// TIA Portal V20 export
FUNCTION_BLOCK "Side_Shifters"   // FB12, LAD
{ S7_Optimized_Access := 'TRUE' }
// stored: MemoryReserve 100, SetENOAutomatically false
   VAR_INPUT
      set_Hydraulic_Up { ExternalAccessible := 'False'; ExternalVisible := 'False'; ExternalWritable := 'False'} : Bool;
      set_Hydraulic_Down { ExternalAccessible := 'False'; ExternalVisible := 'False'; ExternalWritable := 'False'} : Bool;
      set_SL_Hydraulic_Up : Bool;
      set_SL_Hydraulic_Down : Bool;
      set_SR_Hydraulic_Up : Bool;
      set_SR_Hydraulic_Down : Bool;
      set_SL_Hydraulic_Unit : Bool;
      set_SR_Hydraulic_Unit : Bool;
      set_Go_To_ST1 : Bool;
      set_Go_To_ST2 : Bool;
      set_Go_To_ST3 : Bool;
      set_Go_To_ST4 : Bool;
      ST1_Empty : Bool;
      ST2_Empty : Bool;
      ST3_Empty : Bool;
      ST4_Empty : Bool;
      Homing_1_SR : Int;
      Homing_2_SR : Int;
      Homing_3_SR : Int;
      Homing_4_SR : Int;
      Homing_1_SL : Int;
      Homing_2_SL : Int;
      Homing_3_SL : Int;
      Homing_4_SL : Int;
      SL_Drive_Forward : Bool;
      SL_Drive_Backward : Bool;
      SR_Drive_Forward : Bool;
      SR_Drive_Backward : Bool;
      iSL_Sen_Drv_1 : Bool;
      iSL_Sen_Drv_2 : Bool;
      iSL_Sen_Drv_3 : Bool;
      iSL_Sen_Drv_4 : Bool;
      iSR_Sen_Drv_1 : Bool;
      iSR_Sen_Drv_2 : Bool;
      iSR_Sen_Drv_3 : Bool;
      iSR_Sen_Drv_4 : Bool;
      iSL_Sen_Val1_Up : Bool;
      iSL_Sen_Val1_Down : Bool;
      iSL_Sen_Val2_Up : Bool;
      iSL_Sen_Val2_Down : Bool;
      iSR_Sen_Val1_Up : Bool;
      iSR_Sen_Val1_Down : Bool;
      iSR_Sen_Val2_Up : Bool;
      iSR_Sen_Val2_Down : Bool;
      iSL_Distance : Int;
      iSR_Correct : Int;
      iSR_Distance : Int;
      iSL_Hydraulic_Filtr : Bool;
      iSR_Hydraulic_Empty : Bool;
      HWIdentSL : HW_IO;
      HWIdentSR : HW_IO;
      Reset_Drive : Bool;
      Reset_Hydro : Bool;
   END_VAR
   VAR_OUTPUT
      oSL_Valve_Up { ExternalAccessible := 'False'; ExternalVisible := 'False'; ExternalWritable := 'False'} : Bool;
      oSL_Valve_Down { ExternalAccessible := 'False'; ExternalVisible := 'False'; ExternalWritable := 'False'} : Bool;
      oSL_Hydraulic_Unit { ExternalAccessible := 'False'; ExternalVisible := 'False'; ExternalWritable := 'False'} : Bool;
      oSR_Valve_Up { ExternalAccessible := 'False'; ExternalVisible := 'False'; ExternalWritable := 'False'} : Bool;
      oSR_Valve_Down { ExternalAccessible := 'False'; ExternalVisible := 'False'; ExternalWritable := 'False'} : Bool;
      oSR_Hydraulic_Unit { ExternalAccessible := 'False'; ExternalVisible := 'False'; ExternalWritable := 'False'} : Bool;
      oHydraulic_Status_LED_UP_1 : Bool;
      oHydraulic_Status_LED_UP_2 : Bool;
      oHydraulic_Status_LED_DOWN_1 : Bool;
      oHydraulic_Status_LED_DOWN_2 : Bool;
      oSL_Communication_OK : Bool;
      oSR_Communication_OK : Bool;
      oSL_Forward_Flag : Bool;
      oSL_Backward_Flag : Bool;
      oSR_Forward_Flag : Bool;
      oSR_Backward_Flag : Bool;
      oST1_1_Move_Flag : Bool;
      oST1_2_Move_Flag : Bool;
      oST2_1_Move_Flag : Bool;
      oST2_2_Move_Flag : Bool;
      oST3_1_Move_flag : Bool;
      oST3_2_Move_Flag : Bool;
      oST4_1_Move_Flag : Bool;
      oST4_2_Move_Flag : Bool;
   END_VAR
   VAR_IN_OUT
      iSL_Drive_Param : "SEW_MOVIKIT_VelocityDrive_STATUS_V2.1";
      iSR_Drive_Param : "SEW_MOVIKIT_VelocityDrive_STATUS_V2.1";
      oSL_Drive_Param : "SEW_MOVIKIT_VelocityDrive_SETPOINTS_V2.1";
      oSR_Drive_Param : "SEW_MOVIKIT_VelocityDrive_SETPOINTS_V2.1";
   END_VAR
   VAR
      Hydraulic_SL { ExternalAccessible := 'False'; ExternalVisible := 'False'; ExternalWritable := 'False'} : "Side_Hydraulic";
      Hydraulic_SR { ExternalAccessible := 'False'; ExternalVisible := 'False'; ExternalWritable := 'False'} : "Side_Hydraulic";
      Side_Driver_Instance { S7_SetPoint := 'True'} : "Side_Driver";
      Side_Shifter_Auto_Instance { S7_SetPoint := 'True'} : "Side_Shifter_Auto";
      SL_Auto_Speed { S7_SetPoint := 'True'} : Int := 1000;
      SR_Auto_Speed { S7_SetPoint := 'True'} : Int := 1000;
      SL_Auto_Forward : Bool;
      SL_Auto_Backward : Bool;
      SR_Auto_Forward : Bool;
      SR_Auto_Backward : Bool;
      SR_Distance_Correct : Int;
      SL_Error_Laser : Bool;
      SR_Error_Laser : Bool;
      SL_SR_InPosition : Bool;
      SL_Sen_Up : Bool;
      SL_Sen_Down : Bool;
      SR_Sen_Up : Bool;
      SR_Sen_Down : Bool;
      SL_Error_Hyd : Bool;
      SR_Error_Hyd : Bool;
      Error_Drive : Bool;
      Error_Hydro : Bool;
      Status_Sen_Up : Bool;
      Status_Sen_Down : Bool;
      RL_Speed : Int;
      RR_Speed : Int;
      Step_Move_Pallets : Int;
      Row_Start : Int;
      Row_Destination : Int;
      Column_Start : Int;
      Column_Destination : Int;
      TON_iSR_Error { S7_SetPoint := 'True'} : TON_TIME;
      TON_iSL_Error { S7_SetPoint := 'True'} : TON_TIME;
   END_VAR
   VAR_TEMP
      i : SInt;
      FoundIndex : SInt;
   END_VAR
BEGIN

REGION Network 1: Hydraulic control SL
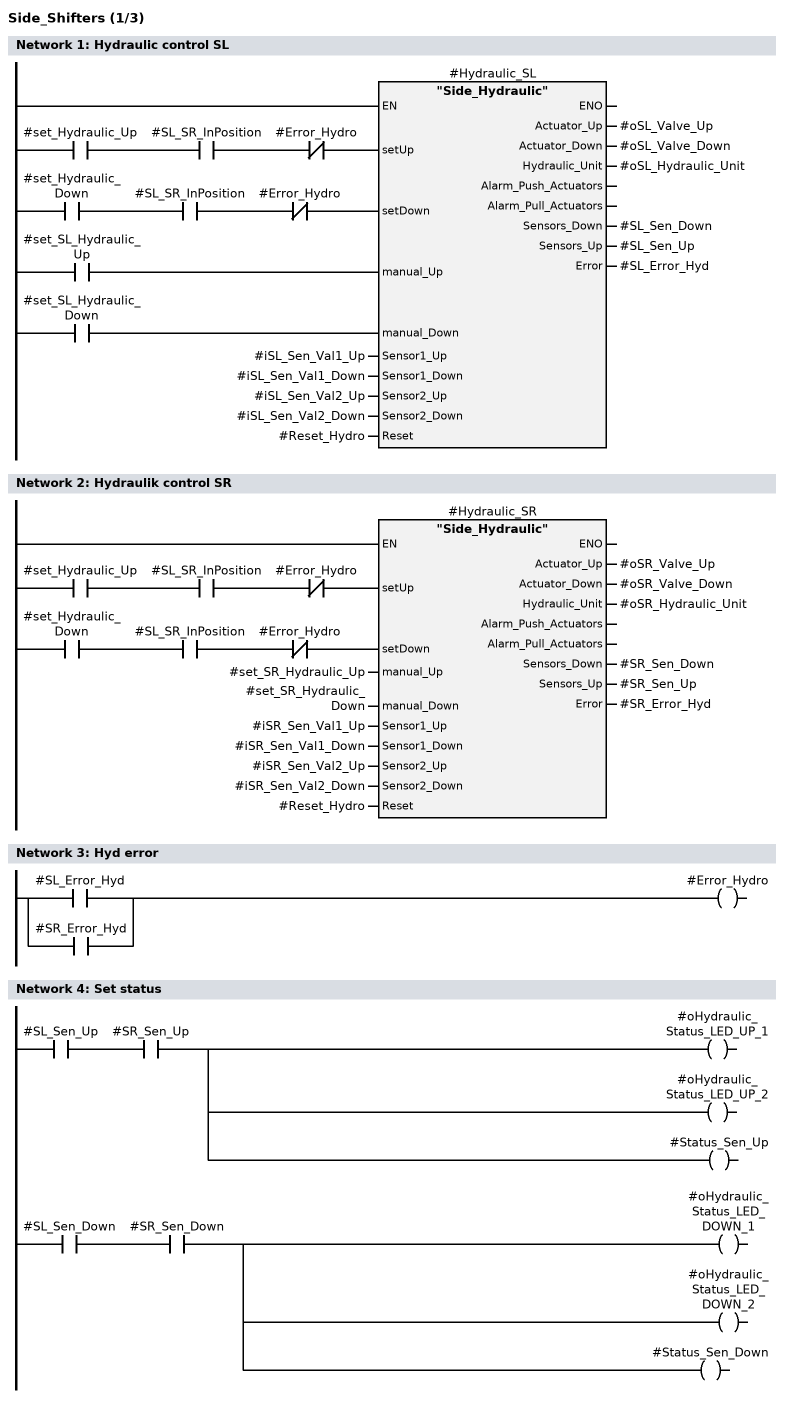
   RUNG wire#powerrail
      #Hydraulic_SL(setUp := wire#w1, setDown := wire#w2, manual_Up := wire#w3, manual_Down := wire#w4, Sensor1_Up := #iSL_Sen_Val1_Up, Sensor1_Down := #iSL_Sen_Val1_Down, Sensor2_Up := #iSL_Sen_Val2_Up, Sensor2_Down := #iSL_Sen_Val2_Down, Reset := #Reset_Hydro, Actuator_Up => #oSL_Valve_Up, Actuator_Down => #oSL_Valve_Down, Hydraulic_Unit => #oSL_Hydraulic_Unit, Alarm_Push_Actuators =>, Alarm_Pull_Actuators =>, Sensors_Down => #SL_Sen_Down, Sensors_Up => #SL_Sen_Up, Error => #SL_Error_Hyd)
   END_RUNG
   RUNG wire#powerrail
      Contact( #set_Hydraulic_Up )
      Contact( #SL_SR_InPosition )
      I_Contact( #Error_Hydro )
   END_RUNG wire#w1
   RUNG wire#powerrail
      Contact( #set_Hydraulic_Down )
      Contact( #SL_SR_InPosition )
      I_Contact( #Error_Hydro )
   END_RUNG wire#w2
   RUNG wire#powerrail
      Contact( #set_SL_Hydraulic_Up )
   END_RUNG wire#w3
   RUNG wire#powerrail
      Contact( #set_SL_Hydraulic_Down )
   END_RUNG wire#w4
   // the same network as SCL:
   #Hydraulic_SL(setUp := #set_Hydraulic_Up AND #SL_SR_InPosition AND NOT #Error_Hydro,   // "Side_Hydraulic"
                 setDown := #set_Hydraulic_Down AND #SL_SR_InPosition AND NOT #Error_Hydro,
                 manual_Up := #set_SL_Hydraulic_Up,
                 manual_Down := #set_SL_Hydraulic_Down,
                 Sensor1_Up := #iSL_Sen_Val1_Up,
                 Sensor1_Down := #iSL_Sen_Val1_Down,
                 Sensor2_Up := #iSL_Sen_Val2_Up,
                 Sensor2_Down := #iSL_Sen_Val2_Down,
                 Reset := #Reset_Hydro,
                 Actuator_Up => #oSL_Valve_Up,
                 Actuator_Down => #oSL_Valve_Down,
                 Hydraulic_Unit => #oSL_Hydraulic_Unit,
                 Sensors_Down => #SL_Sen_Down,
                 Sensors_Up => #SL_Sen_Up,
                 Error => #SL_Error_Hyd);
END_REGION

REGION Network 2: Hydraulik control SR
   RUNG wire#powerrail
      #Hydraulic_SR(setUp := wire#w1, setDown := wire#w2, manual_Up := #set_SR_Hydraulic_Up, manual_Down := #set_SR_Hydraulic_Down, Sensor1_Up := #iSR_Sen_Val1_Up, Sensor1_Down := #iSR_Sen_Val1_Down, Sensor2_Up := #iSR_Sen_Val2_Up, Sensor2_Down := #iSR_Sen_Val2_Down, Reset := #Reset_Hydro, Actuator_Up => #oSR_Valve_Up, Actuator_Down => #oSR_Valve_Down, Hydraulic_Unit => #oSR_Hydraulic_Unit, Alarm_Push_Actuators =>, Alarm_Pull_Actuators =>, Sensors_Down => #SR_Sen_Down, Sensors_Up => #SR_Sen_Up, Error => #SR_Error_Hyd)
   END_RUNG
   RUNG wire#powerrail
      Contact( #set_Hydraulic_Up )
      Contact( #SL_SR_InPosition )
      I_Contact( #Error_Hydro )
   END_RUNG wire#w1
   RUNG wire#powerrail
      Contact( #set_Hydraulic_Down )
      Contact( #SL_SR_InPosition )
      I_Contact( #Error_Hydro )
   END_RUNG wire#w2
   // the same network as SCL:
   #Hydraulic_SR(setUp := #set_Hydraulic_Up AND #SL_SR_InPosition AND NOT #Error_Hydro,   // "Side_Hydraulic"
                 setDown := #set_Hydraulic_Down AND #SL_SR_InPosition AND NOT #Error_Hydro,
                 manual_Up := #set_SR_Hydraulic_Up,
                 manual_Down := #set_SR_Hydraulic_Down,
                 Sensor1_Up := #iSR_Sen_Val1_Up,
                 Sensor1_Down := #iSR_Sen_Val1_Down,
                 Sensor2_Up := #iSR_Sen_Val2_Up,
                 Sensor2_Down := #iSR_Sen_Val2_Down,
                 Reset := #Reset_Hydro,
                 Actuator_Up => #oSR_Valve_Up,
                 Actuator_Down => #oSR_Valve_Down,
                 Hydraulic_Unit => #oSR_Hydraulic_Unit,
                 Sensors_Down => #SR_Sen_Down,
                 Sensors_Up => #SR_Sen_Up,
                 Error => #SR_Error_Hyd);
END_REGION

REGION Network 3: Hyd error
   RUNG wire#powerrail
      Contact( #SL_Error_Hyd )
      wire#w1
      Coil( #Error_Hydro )
   END_RUNG
   RUNG wire#powerrail
      Contact( #SR_Error_Hyd )
   END_RUNG wire#w1
   // the same network as SCL:
   #Error_Hydro := #SL_Error_Hyd OR #SR_Error_Hyd;
END_REGION

REGION Network 4: Set status
   RUNG wire#powerrail
      Contact( #SL_Sen_Up )
      Contact( #SR_Sen_Up )
      wire#w1
      Coil( #oHydraulic_Status_LED_UP_1 )
   END_RUNG
   RUNG wire#w1
      Coil( #oHydraulic_Status_LED_UP_2 )
   END_RUNG
   RUNG wire#w1
      Coil( #Status_Sen_Up )
   END_RUNG
   RUNG wire#powerrail
      Contact( #SL_Sen_Down )
      Contact( #SR_Sen_Down )
      wire#w2
      Coil( #oHydraulic_Status_LED_DOWN_1 )
   END_RUNG
   RUNG wire#w2
      Coil( #oHydraulic_Status_LED_DOWN_2 )
   END_RUNG
   RUNG wire#w2
      Coil( #Status_Sen_Down )
   END_RUNG
   // the same network as SCL:
   #oHydraulic_Status_LED_UP_1 := #SL_Sen_Up AND #SR_Sen_Up;
   #oHydraulic_Status_LED_UP_2 := #oHydraulic_Status_LED_UP_1;
   #Status_Sen_Up := #oHydraulic_Status_LED_UP_1;
   #oHydraulic_Status_LED_DOWN_1 := #SL_Sen_Down AND #SR_Sen_Down;
   #oHydraulic_Status_LED_DOWN_2 := #oHydraulic_Status_LED_DOWN_1;
   #Status_Sen_Down := #oHydraulic_Status_LED_DOWN_1;
END_REGION

REGION Network 5: Make correct on SR distance
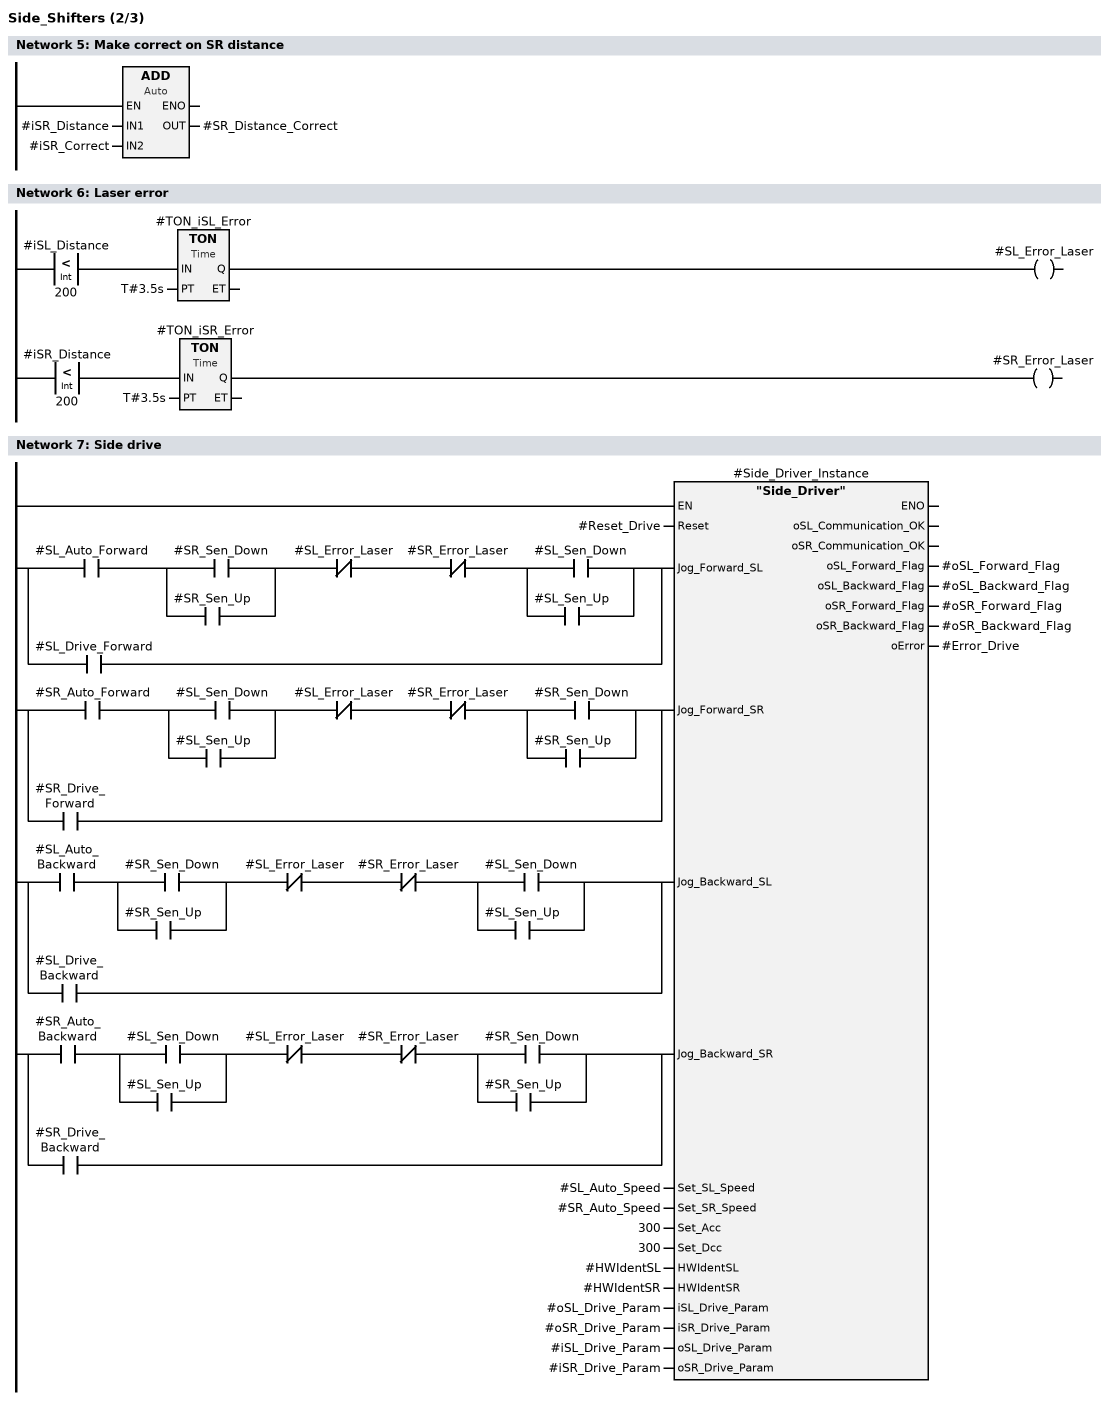
   RUNG wire#powerrail
      Add(in1 := #iSR_Distance, in2 := #iSR_Correct, out => #SR_Distance_Correct)
   END_RUNG
   // the same network as SCL:
   #SR_Distance_Correct := #iSR_Distance + #iSR_Correct;
END_REGION

REGION Network 6: Laser error
   RUNG wire#powerrail
      { S7_Templates := "SrcType := Int" } LT_Contact(in1 := #iSL_Distance, in2 := 200)
      { S7_Templates := "time_type := Time" } #TON_iSL_Error.TON(pt := T#3.5s, et =>)
      Coil( #SL_Error_Laser )
   END_RUNG
   RUNG wire#powerrail
      { S7_Templates := "SrcType := Int" } LT_Contact(in1 := #iSR_Distance, in2 := 200)
      { S7_Templates := "time_type := Time" } #TON_iSR_Error.TON(pt := T#3.5s, et =>)
      Coil( #SR_Error_Laser )
   END_RUNG
   // the same network as SCL:
   #TON_iSL_Error(IN := #iSL_Distance < 200, PT := T#3.5s);   // TON
   #SL_Error_Laser := #TON_iSL_Error.Q;
   #TON_iSR_Error(IN := #iSR_Distance < 200, PT := T#3.5s);   // TON
   #SR_Error_Laser := #TON_iSR_Error.Q;
END_REGION

REGION Network 7: Side drive
   RUNG wire#powerrail
      #Side_Driver_Instance(Jog_Forward_SL := wire#w4, Jog_Forward_SR := wire#w8, Jog_Backward_SL := wire#w12, Jog_Backward_SR := wire#w16, Reset := #Reset_Drive, Set_SL_Speed := #SL_Auto_Speed, Set_SR_Speed := #SR_Auto_Speed, Set_Acc := 300, Set_Dcc := 300, HWIdentSL := #HWIdentSL, HWIdentSR := #HWIdentSR, iSL_Drive_Param := #oSL_Drive_Param, iSR_Drive_Param := #oSR_Drive_Param, oSL_Drive_Param := #iSL_Drive_Param, oSR_Drive_Param := #iSR_Drive_Param, oSL_Communication_OK =>, oSR_Communication_OK =>, oSL_Forward_Flag => #oSL_Forward_Flag, oSL_Backward_Flag => #oSL_Backward_Flag, oSR_Forward_Flag => #oSR_Forward_Flag, oSR_Backward_Flag => #oSR_Backward_Flag, oError => #Error_Drive)
   END_RUNG
   RUNG wire#powerrail
      Contact( #SL_Auto_Forward )
      wire#w1
      Contact( #SR_Sen_Down )
      wire#w2
      I_Contact( #SL_Error_Laser )
      I_Contact( #SR_Error_Laser )
      wire#w3
      Contact( #SL_Sen_Down )
   END_RUNG wire#w4
   RUNG wire#w1
      Contact( #SR_Sen_Up )
   END_RUNG wire#w2
   RUNG wire#w3
      Contact( #SL_Sen_Up )
   END_RUNG wire#w4
   RUNG wire#powerrail
      Contact( #SL_Drive_Forward )
   END_RUNG wire#w4
   RUNG wire#powerrail
      Contact( #SR_Auto_Forward )
      wire#w5
      Contact( #SL_Sen_Down )
      wire#w6
      I_Contact( #SL_Error_Laser )
      I_Contact( #SR_Error_Laser )
      wire#w7
      Contact( #SR_Sen_Down )
   END_RUNG wire#w8
   RUNG wire#w5
      Contact( #SL_Sen_Up )
   END_RUNG wire#w6
   RUNG wire#w7
      Contact( #SR_Sen_Up )
   END_RUNG wire#w8
   RUNG wire#powerrail
      Contact( #SR_Drive_Forward )
   END_RUNG wire#w8
   RUNG wire#powerrail
      Contact( #SL_Auto_Backward )
      wire#w9
      Contact( #SR_Sen_Down )
      wire#w10
      I_Contact( #SL_Error_Laser )
      I_Contact( #SR_Error_Laser )
      wire#w11
      Contact( #SL_Sen_Down )
   END_RUNG wire#w12
   RUNG wire#w9
      Contact( #SR_Sen_Up )
   END_RUNG wire#w10
   RUNG wire#w11
      Contact( #SL_Sen_Up )
   END_RUNG wire#w12
   RUNG wire#powerrail
      Contact( #SL_Drive_Backward )
   END_RUNG wire#w12
   RUNG wire#powerrail
      Contact( #SR_Auto_Backward )
      wire#w13
      Contact( #SL_Sen_Down )
      wire#w14
      I_Contact( #SL_Error_Laser )
      I_Contact( #SR_Error_Laser )
      wire#w15
      Contact( #SR_Sen_Down )
   END_RUNG wire#w16
   RUNG wire#w13
      Contact( #SL_Sen_Up )
   END_RUNG wire#w14
   RUNG wire#w15
      Contact( #SR_Sen_Up )
   END_RUNG wire#w16
   RUNG wire#powerrail
      Contact( #SR_Drive_Backward )
   END_RUNG wire#w16
   // the same network as SCL:
   #Side_Driver_Instance(Reset := #Reset_Drive,   // "Side_Driver"
                         Jog_Forward_SL := (#SL_Auto_Forward AND (#SR_Sen_Down OR #SR_Sen_Up) AND NOT #SL_Error_Laser AND NOT #SR_Error_Laser AND (#SL_Sen_Down OR #SL_Sen_Up)) OR #SL_Drive_Forward,
                         Jog_Forward_SR := (#SR_Auto_Forward AND (#SL_Sen_Down OR #SL_Sen_Up) AND NOT #SL_Error_Laser AND NOT #SR_Error_Laser AND (#SR_Sen_Down OR #SR_Sen_Up)) OR #SR_Drive_Forward,
                         Jog_Backward_SL := (#SL_Auto_Backward AND (#SR_Sen_Down OR #SR_Sen_Up) AND NOT #SL_Error_Laser AND NOT #SR_Error_Laser AND (#SL_Sen_Down OR #SL_Sen_Up)) OR #SL_Drive_Backward,
                         Jog_Backward_SR := (#SR_Auto_Backward AND (#SL_Sen_Down OR #SL_Sen_Up) AND NOT #SL_Error_Laser AND NOT #SR_Error_Laser AND (#SR_Sen_Down OR #SR_Sen_Up)) OR #SR_Drive_Backward,
                         Set_SL_Speed := #SL_Auto_Speed,
                         Set_SR_Speed := #SR_Auto_Speed,
                         Set_Acc := 300,
                         Set_Dcc := 300,
                         HWIdentSL := #HWIdentSL,
                         HWIdentSR := #HWIdentSR,
                         iSL_Drive_Param := #oSL_Drive_Param,
                         iSR_Drive_Param := #oSR_Drive_Param,
                         oSL_Drive_Param := #iSL_Drive_Param,
                         oSR_Drive_Param := #iSR_Drive_Param,
                         oSL_Forward_Flag => #oSL_Forward_Flag,
                         oSL_Backward_Flag => #oSL_Backward_Flag,
                         oSR_Forward_Flag => #oSR_Forward_Flag,
                         oSR_Backward_Flag => #oSR_Backward_Flag,
                         oError => #Error_Drive);
END_REGION

REGION Network 8: Auto moving
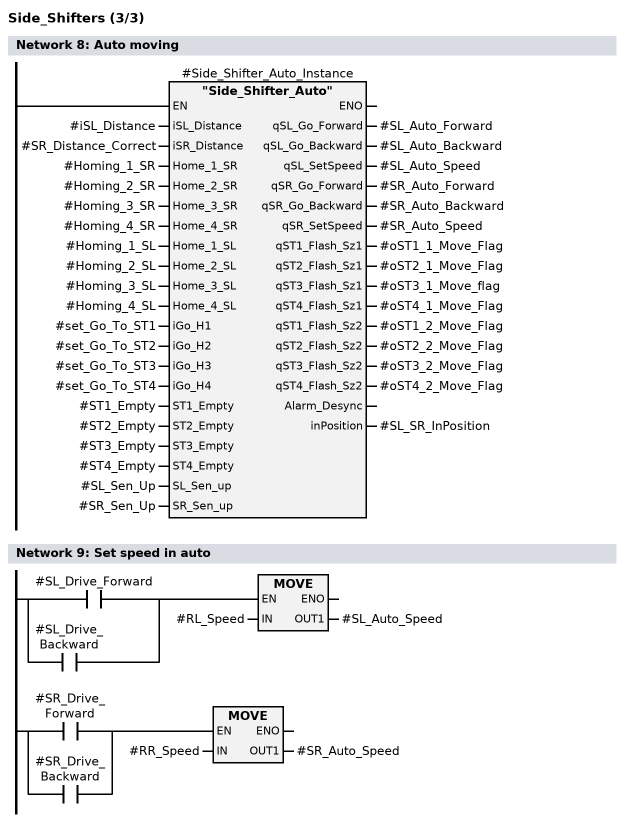
   RUNG wire#powerrail
      #Side_Shifter_Auto_Instance(iSL_Distance := #iSL_Distance, iSR_Distance := #SR_Distance_Correct, Home_1_SR := #Homing_1_SR, Home_2_SR := #Homing_2_SR, Home_3_SR := #Homing_3_SR, Home_4_SR := #Homing_4_SR, Home_1_SL := #Homing_1_SL, Home_2_SL := #Homing_2_SL, Home_3_SL := #Homing_3_SL, Home_4_SL := #Homing_4_SL, iGo_H1 := #set_Go_To_ST1, iGo_H2 := #set_Go_To_ST2, iGo_H3 := #set_Go_To_ST3, iGo_H4 := #set_Go_To_ST4, ST1_Empty := #ST1_Empty, ST2_Empty := #ST2_Empty, ST3_Empty := #ST3_Empty, ST4_Empty := #ST4_Empty, SL_Sen_up := #SL_Sen_Up, SR_Sen_up := #SR_Sen_Up, qSL_Go_Forward => #SL_Auto_Forward, qSL_Go_Backward => #SL_Auto_Backward, qSL_SetSpeed => #SL_Auto_Speed, qSR_Go_Forward => #SR_Auto_Forward, qSR_Go_Backward => #SR_Auto_Backward, qSR_SetSpeed => #SR_Auto_Speed, qST1_Flash_Sz1 => #oST1_1_Move_Flag, qST2_Flash_Sz1 => #oST2_1_Move_Flag, qST3_Flash_Sz1 => #oST3_1_Move_flag, qST4_Flash_Sz1 => #oST4_1_Move_Flag, qST1_Flash_Sz2 => #oST1_2_Move_Flag, qST2_Flash_Sz2 => #oST2_2_Move_Flag, qST3_Flash_Sz2 => #oST3_2_Move_Flag, qST4_Flash_Sz2 => #oST4_2_Move_Flag, Alarm_Desync =>, inPosition => #SL_SR_InPosition)
   END_RUNG
   // the same network as SCL:
   #Side_Shifter_Auto_Instance(iSL_Distance := #iSL_Distance,   // "Side_Shifter_Auto"
                           iSR_Distance := #SR_Distance_Correct,
                           Home_1_SR := #Homing_1_SR,
                           Home_2_SR := #Homing_2_SR,
                           Home_3_SR := #Homing_3_SR,
                           Home_4_SR := #Homing_4_SR,
                           Home_1_SL := #Homing_1_SL,
                           Home_2_SL := #Homing_2_SL,
                           Home_3_SL := #Homing_3_SL,
                           Home_4_SL := #Homing_4_SL,
                           iGo_H1 := #set_Go_To_ST1,
                           iGo_H2 := #set_Go_To_ST2,
                           iGo_H3 := #set_Go_To_ST3,
                           iGo_H4 := #set_Go_To_ST4,
                           ST1_Empty := #ST1_Empty,
                           ST2_Empty := #ST2_Empty,
                           ST3_Empty := #ST3_Empty,
                           ST4_Empty := #ST4_Empty,
                           SL_Sen_up := #SL_Sen_Up,
                           SR_Sen_up := #SR_Sen_Up,
                           qSL_Go_Forward => #SL_Auto_Forward,
                           qSL_Go_Backward => #SL_Auto_Backward,
                           qSL_SetSpeed => #SL_Auto_Speed,
                           qSR_Go_Forward => #SR_Auto_Forward,
                           qSR_Go_Backward => #SR_Auto_Backward,
                           qSR_SetSpeed => #SR_Auto_Speed,
                           qST1_Flash_Sz1 => #oST1_1_Move_Flag,
                           qST2_Flash_Sz1 => #oST2_1_Move_Flag,
                           qST3_Flash_Sz1 => #oST3_1_Move_flag,
                           qST4_Flash_Sz1 => #oST4_1_Move_Flag,
                           qST1_Flash_Sz2 => #oST1_2_Move_Flag,
                           qST2_Flash_Sz2 => #oST2_2_Move_Flag,
                           qST3_Flash_Sz2 => #oST3_2_Move_Flag,
                           qST4_Flash_Sz2 => #oST4_2_Move_Flag,
                           inPosition => #SL_SR_InPosition);
END_REGION

REGION Network 9: Set speed in auto
   RUNG wire#powerrail
      Contact( #SL_Drive_Forward )
      wire#w1
      Move(in := #RL_Speed, out1 => #SL_Auto_Speed)
   END_RUNG
   RUNG wire#powerrail
      Contact( #SL_Drive_Backward )
   END_RUNG wire#w1
   RUNG wire#powerrail
      Contact( #SR_Drive_Forward )
      wire#w2
      Move(in := #RR_Speed, out1 => #SR_Auto_Speed)
   END_RUNG
   RUNG wire#powerrail
      Contact( #SR_Drive_Backward )
   END_RUNG wire#w2
   // the same network as SCL:
   IF #SL_Drive_Forward OR #SL_Drive_Backward THEN #SL_Auto_Speed := #RL_Speed; END_IF;
   IF #SR_Drive_Forward OR #SR_Drive_Backward THEN #SR_Auto_Speed := #RR_Speed; END_IF;
END_REGION

REGION Network 10 (SCL): SS1 - Move Pallet
   IF #HWIdentSL = "S1R1M~Module_I_O_(05_words)_1" THEN

       IF (#Hydraulic_SL.Actuator_Up OR #Hydraulic_SR.Actuator_Up) AND #Status_Sen_Up AND #Step_Move_Pallets = 0 THEN
           #Step_Move_Pallets := 1;
           IF #oST1_1_Move_Flag THEN
               #Row_Start := 1;
               #Column_Start := 11;
           ELSIF #oST2_1_Move_Flag THEN
               #Row_Start := 2;
               #Column_Start := 12;
           ELSIF #oST3_1_Move_flag THEN
               #Row_Start := 3;
               #Column_Start := 11;
           ELSIF #oST4_1_Move_Flag THEN
               #Row_Start := 4;
               #Column_Start := 11;
           END_IF;

       ELSIF (#Hydraulic_SL.Actuator_Down OR #Hydraulic_SR.Actuator_Down) AND #Status_Sen_Up AND #Step_Move_Pallets = 1 THEN
           #Step_Move_Pallets := 2;
           IF #oST1_1_Move_Flag THEN
               #Row_Destination := 1;
               #Column_Destination := 11;
           ELSIF #oST2_1_Move_Flag THEN
               #Row_Destination := 2;
               #Column_Destination := 12;
           ELSIF #oST3_1_Move_flag THEN
               #Row_Destination := 3;
               #Column_Destination := 11;
           ELSIF #oST4_1_Move_Flag THEN
               #Row_Destination := 4;
               #Column_Destination := 11;
           END_IF;

       ELSIF #Step_Move_Pallets = 2 THEN
           FOR #i := 1 TO 24 DO
               IF ("Pallets_Stations".Pallets[#i].Station_Current_Position[1] = #Row_Start) AND
                   ("Pallets_Stations".Pallets[#i].Station_Current_Position[2] = #Column_Start) THEN
                   #FoundIndex := #i;
                   EXIT;
               END_IF;
           END_FOR;

           IF #FoundIndex <> 0 THEN
               "Pallets_Stations".Pallets[#FoundIndex].Station_Current_Position[1] := #Row_Destination;
               "Pallets_Stations".Pallets[#FoundIndex].Station_Current_Position[2] := #Column_Destination;
           END_IF;
           #Step_Move_Pallets := 0;

       END_IF;
   END_IF;
END_REGION

REGION Network 11 (SCL): SS2 - Move Pallet
   IF #HWIdentSL = "S2R2M~Module_I_O_(05_words)_1" THEN
       #Column_Start := 1;
       IF (#Hydraulic_SL.Actuator_Up OR #Hydraulic_SR.Actuator_Up) AND #Status_Sen_Up AND #Step_Move_Pallets = 0 THEN
           #Step_Move_Pallets := 1;
           IF #oST1_1_Move_Flag THEN
               #Row_Start := 1;
           ELSIF #oST2_1_Move_Flag THEN
               #Row_Start := 2;
           ELSIF #oST3_1_Move_flag THEN
               #Row_Start := 3;
           ELSIF #oST4_1_Move_Flag THEN
               #Row_Start := 4;
           END_IF;

       ELSIF (#Hydraulic_SL.Actuator_Down OR #Hydraulic_SR.Actuator_Down) AND #Status_Sen_Up AND #Step_Move_Pallets = 1 THEN
           #Step_Move_Pallets := 2;
           IF #oST1_1_Move_Flag THEN
               #Row_Destination := 1;
           ELSIF #oST2_1_Move_Flag THEN
               #Row_Destination := 2;
           ELSIF #oST3_1_Move_flag THEN
               #Row_Destination := 3;
           ELSIF #oST4_1_Move_Flag THEN
               #Row_Destination := 4;
           END_IF;

       ELSIF #Step_Move_Pallets = 2 THEN
           FOR #i := 1 TO 24 DO
               IF ("Pallets_Stations".Pallets[#i].Station_Current_Position[1] = #Row_Start) AND
                   ("Pallets_Stations".Pallets[#i].Station_Current_Position[2] = #Column_Start) THEN
                   #FoundIndex := #i;
                   EXIT;
               END_IF;
           END_FOR;

           IF #FoundIndex <> 0 THEN
               "Pallets_Stations".Pallets[#FoundIndex].Station_Current_Position[1] := #Row_Destination;
               "Pallets_Stations".Pallets[#FoundIndex].Station_Current_Position[2] := #Column_Destination;
           END_IF;
           #Step_Move_Pallets := 0;

       END_IF;
   END_IF;
END_REGION
END_FUNCTION_BLOCK
